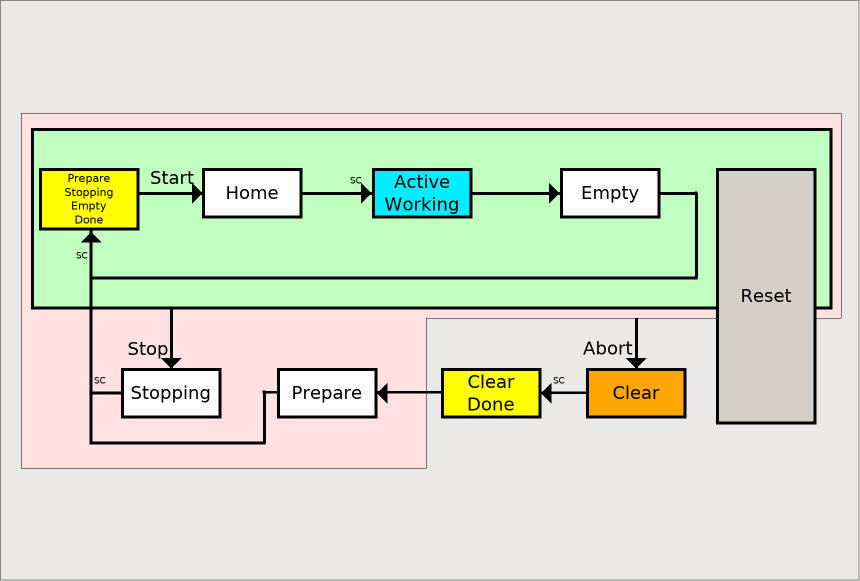
VISUALIZATION FrameXtsStateModel  // 860x581
VAR_IN_OUT

	eOPMState			: E_OperatingState;
	eStateCommand		: E_OperatingCmd;
	
END_VAR
    Rectangle (-10,1 860x580)
    Polygon (21,113) (841,113) (841,318) (426,318) (426,468) (21,468)
    Rectangle (31,128 801x181)
    Polyline (636,318) (636,393) (264,392) (264,443) (191,443) (91,443) (91,393) (91,193) (411,193)
    RoundedRectangle (39,168 100x62), "Prepare Stopping Empty Done", colour toggle: eOPMState = E_OperatingState.OperatingMode_Prepar_Sc
    RoundedRectangle (202,168 100x50), "Home", colour toggle: (eOPMState = E_OperatingState.OperatingMode_Home)
        OnMouseClick: execute { eStateCommand := E_OperatingCmd.OperatingCmd_Home; }
    RoundedRectangle (277,368 100x50), "Prepare", colour toggle: (eOPMState = E_OperatingState.OperatingMode_Prepare)
        OnMouseClick: execute { eStateCommand := E_OperatingCmd.OperatingCmd_Prepare; }
    RoundedRectangle (441,368 100x50), "Clear Done", colour toggle: (eOPMState = E_OperatingState.OperatingMode_Clear_Sc)
    RoundedRectangle (586,368 100x50), "Clear", colour toggle: (eOPMState = E_OperatingState.OperatingMode_Clear)
        OnMouseClick: execute { eStateCommand := E_OperatingCmd.OperatingCmd_Clear; }
    Polygon (91,232) (81,242) (101,242)
    Polygon (541,393) (551,403) (551,383)
    Polygon (377,393) (387,403) (387,383)
    Polygon (202,193) (192,203) (192,183)
    Polygon (371,193) (361,203) (361,183)
    Polygon (559,193) (549,203) (549,183)
    Polygon (646,358) (636,368) (626,358)
    Polygon (181,358) (171,368) (161,358)
    Polyline (171,308) (171,393) (91,393)
    RoundedRectangle (121,368 100x50), "Stopping", colour toggle: (eOPMState = E_OperatingState.OperatingMode_Stopping)
        OnMouseClick: execute { eStateCommand := E_OperatingCmd.OperatingCmd_Stopping; }
    Label (316,173 80x15), "SC"
    Polyline (396,193) (696,193) (696,278) (92,278)
    Label (519,373 80x15), "SC"
    Label (60,373 80x15), "SC"
    Label (108,339 80x20), "Stop"
    Label (568,339 80x19), "Abort"
    Label (42,248 80x15), "SC"
    Label (132,169 80x18), "Start", invisible if: eOPMState <> E_OperatingState.OperatingMode_Prepar_Sc
    RoundedRectangle (560,168 100x50), "Empty", colour toggle: (eOPMState = E_OperatingState.OperatingMode_Empty)
        OnMouseClick: execute { eStateCommand := E_OperatingCmd.OperatingCmd_Empty; }
    RoundedRectangle (716,168 100x256), "Reset", colour toggle: (eOPMState = E_OperatingState.OperatingMode_Reset)
        OnMouseClick: execute { eStateCommand := E_OperatingCmd.OperatingCmd_Reset; }
    RoundedRectangle (372,168 100x50), "Active Working", colour toggle: (eOPMState = E_OperatingState.OperatingMode_Active)
END_VISUALIZATION

(* stored: Version 1.1.0.1, ProductVersion 3.1.4024.12
   Visu FrameXtsStateModel: Id {4cf49023-0575-4d13-ac94-deebcaff7985} *)
